// TIA Portal V19 export
VAR_GLOBAL   // PLC tag table "Default tag table"
   Tag_40 AT %T82 : Timer;
   Tag_41 AT %M19.7 : Bool;
   Tag_42 AT %M20.5 : Bool;
   Tag_43 AT %T115 : Timer;
   Tag_44 AT %T114 : Timer;
   Tag_45 AT %T148 : Timer;
   Tag_46 AT %T116 : Timer;
   Tag_47 AT %T117 : Timer;
   Tag_48 AT %T149 : Timer;
   Tag_49 AT %M13.0 : Bool;
   Tag_50 AT %MB210 : Byte;
   Tag_51 AT %MB213 : Byte;
   Tag_52 AT %MB211 : Byte;
   Tag_53 AT %MB212 : Byte;
   Tag_54 AT %T68 : Timer;
   Tag_55 AT %T56 : Timer;
   Tag_56 AT %T80 : Timer;
   Tag_57 AT %M30.0 : Bool;
   Tag_58 AT %T10 : Timer;
   Tag_59 AT %T11 : Timer;
   Tag_60 AT %T12 : Timer;
   Tag_61 AT %T13 : Timer;
   Tag_62 AT %T19 : Timer;
   Tag_63 AT %T21 : Timer;
   Tag_64 AT %T22 : Timer;
   Tag_65 AT %T23 : Timer;
   Tag_66 AT %T24 : Timer;
   Tag_67 AT %T25 : Timer;
   Tag_68 AT %T26 : Timer;
   Tag_69 AT %T57 : Timer;
   Tag_70 AT %T62 : Timer;
   Tag_71 AT %T63 : Timer;
   Tag_72 AT %T64 : Timer;
   Tag_73 AT %T65 : Timer;
   Tag_74 AT %M152.7 : Bool;
   Tag_75 AT %MW222 : Word;
   Tag_76 AT %MW230 : Word;
   Tag_77 AT %M1.0 : Bool;
   Tag_78 AT %T69 : Timer;
   Tag_79 AT %M19.6 : Bool;
   Tag_80 AT %T81 : Timer;
   Tag_81 AT %Q535.0 : Bool;
   Tag_82 AT %IW12 : Word;
   Tag_83 AT %IW16 : Word;
   Tag_84 AT %IW24 : Word;
   Tag_85 AT %IW32 : Word;
   Tag_86 AT %IW44 : Word;
   Tag_87 AT %IW46 : Word;
   Tag_88 AT %MW84 : Word;
   Tag_89 AT %MW94 : Word;
   Tag_90 AT %MW98 : Word;
   Tag_91 AT %T100 : Timer;
   Tag_92 AT %T101 : Timer;
   Tag_93 AT %T102 : Timer;
   Tag_94 AT %M132.0 : Bool;
   Tag_95 AT %M132.1 : Bool;
   Tag_96 AT %M132.2 : Bool;
   Tag_97 AT %M132.3 : Bool;
   Tag_98 AT %M132.4 : Bool;
   Tag_99 AT %T58 : Timer;
   Tag_100 AT %T59 : Timer;
   Tag_101 AT %T103 : Timer;
   Tag_102 AT %T104 : Timer;
   Tag_103 AT %T105 : Timer;
   Tag_104 AT %M15.1 : Bool;
   Tag_105 AT %M15.2 : Bool;
   Tag_106 AT %T106 : Timer;
   Tag_107 AT %T107 : Timer;
   Tag_108 AT %T71 : Timer;
   Tag_109 AT %T72 : Timer;
   Tag_110 AT %M20.1 : Bool;
   Tag_111 AT %T108 : Timer;
   Tag_112 AT %T109 : Timer;
   Tag_113 AT %T110 : Timer;
   Tag_114 AT %T111 : Timer;
   Tag_115 AT %T112 : Timer;
   Tag_116 AT %T113 : Timer;
   Tag_117 AT %T118 : Timer;
   Tag_118 AT %T93 : Timer;
   Tag_119 AT %M141.0 : Bool;
   Tag_120 AT %M141.1 : Bool;
   Tag_121 AT %M141.2 : Bool;
   Tag_122 AT %M144.1 : Bool;
END_VAR
VAR_GLOBAL CONSTANT   // user constants
   Y0101_ : Int := 1;
   Y0103_ : Int := 2;
   Y0104_ : Int := 3;
   Y0109_ : Int := 4;
   Y0111_ : Int := 5;
   Y0112_ : Int := 6;
   Y0113_ : Int := 7;
   Y0114_ : Int := 8;
   Y0115_ : Int := 9;
   M0139_ : Int := 10;
   Y0116_ : Int := 11;
   Y0108_ : Int := 12;
   Y0117_ : Int := 13;
   Y0118_ : Int := 14;
   Y0237_ : Int := 15;
   Y0238_ : Int := 16;
   Y0119_ : Int := 17;
   Y0124_ : Int := 18;
   Y0135_NOT_USED_ : Int := 19;
   Y0136_NOT_USED_ : Int := 20;
   Y0137_NOT_USED_ : Int := 21;
   Y0143_ : Int := 22;
   Y0144_NOT_USED_ : Int := 23;
   Y0147_ : Int := 24;
   Y0148_ : Int := 25;
   Y0158_ : Int := 26;
   Y0545_ : Int := 27;
   PACK1_ : Int := 28;
   PACK2_ : Int := 29;
   PACK3_ : Int := 30;
   PACK4_ : Int := 31;
   AlarmLamp_ : Int := 32;
   AHV_CLOSED_ : Int := 33;
   AHV_HIGH_LEVEL_ : Int := 34;
   AHV_READY_ : Int := 35;
   AHV_SHUT_DOWN_ : Int := 36;
   AHV_STERILE_ : Int := 37;
   PROD_AVAILABLE_ : Int := 38;
   RINSE_READY_ : Int := 39;
   CAUSTIC_READY_ : Int := 40;
   ACID_READY_ : Int := 41;
   CIP_FILLER_ENABLE_ : Int := 42;
   WATER_PUMP_ : Int := 43;
   Y0901_ : Int := 44;
   Y0902_ : Int := 45;
   Y0903_ : Int := 46;
   TANK_READY_ : Int := 47;
   TANK_OPEN_ : Int := 48;
   Y0904_ : Int := 49;
   Y0905_ : Int := 50;
   Y0906_ : Int := 51;
   Y0907_ : Int := 52;
   Y0908_ : Int := 53;
   Y0909_ : Int := 54;
   Y0910_ : Int := 55;
   Y0911_ : Int := 56;
   Y0912_ : Int := 57;
   Q41_1_ : Int := 58;
   CIP_Route_ : Int := 59;
   SIP_Steam_ : Int := 60;
   Product_Available_ : Int := 61;
   Barrier_Sterile_ : Int := 62;
   Product_Route_ : Int := 63;
   X0913_ : Int := 64;
   V0930_ : Int := 65;
   V0931_ : Int := 66;
   spare2_ : Int := 67;
   V0552_ : Int := 68;
   V0934_ : Int := 69;
   V0935_ : Int := 70;
   V0940_ : Int := 71;
   V0941_ : Int := 72;
   V0942_ : Int := 73;
   V0943_ : Int := 74;
   V0944_ : Int := 75;
   V0945_ : Int := 76;
   M0940_ : Int := 77;
   V1021_ : Int := 78;
   V1023_ : Int := 79;
   V1024_ : Int := 80;
   V1025_ : Int := 81;
   V1027_ : Int := 82;
   V1083_ : Int := 83;
   M0941_ : Int := 84;
   V0936_ : Int := 85;
END_VAR
